(* PLC project Programme MGS_2-07_refactorJOY.project, CODESYS CODESYS V3.5 SP19 Patch 1 *)
(* stored: creationDateTime 2026-06-29T23:37:38.6365562, modificationDateTime 2026-06-29T22:49:33.424 *)

PROGRAM PROGRAMME_IP

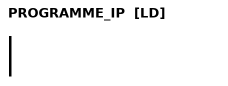
(* LD diagram, written out as Structured Text *)
END_PROGRAM
